TYPE ST_UserControl_Manual_Device_FromHmi :
STRUCT
	stOn,
	stOff		: ST_HMI_BUTTON_IN;	
END_STRUCT
END_TYPE

(* stored: Version 1.1.0.1, ProductVersion 3.1.4024.11
   DUT ST_UserControl_Manual_Device_FromHmi: Id {d0ae3481-964b-450c-aef8-858dac700fa9} *)
